// TIA Portal project "FactoryIO_Template_S7-1200_V15" (V15)
// Vorlageprojekt für das Buch mit Zielsystem S7-1200

(* hardware
DEVICE "S7-1200-Station_1"  S7-1200 Station
   slot 0: "Baugruppenträger_0"  Rack  V1.0
   slot 1: "PLC_1"  CPU 1211C DC/DC/DC  6ES7 211-1AE40-0XB0  V4.1
*)

// ===== PLC "PLC_1"  CPU 1211C DC/DC/DC =====

VAR_GLOBAL   // PLC tag table "Standard-Variablentabelle"
   "START" AT %I0.0 : Bool;
   "STOP" AT %I0.1 : Bool;
   "SENSOR 1" AT %I0.2 : Bool;
   "SENSOR 2" AT %I0.3 : Bool;
   "SENSOR 3" AT %I0.4 : Bool;
   "SENSOR 4" AT %I0.5 : Bool;
   "BELT 6m" AT %Q0.0 : Bool;
   "BELT 4m 1" AT %Q0.1 : Bool;
   "BELT 4m 2" AT %Q0.2 : Bool;
   "BELT 4m 3" AT %Q0.3 : Bool;
   "Wheel Right" AT %Q0.4 : Bool;
   "Wheel Left" AT %Q0.5 : Bool;
   "Wheel Forwerd" AT %Q0.6 : Bool;
   "Working" AT %Q0.7 : Bool;
   "Stoped" AT %Q1.0 : Bool;
   "X" AT %M0.0 : Bool;
   "Y" AT %M0.1 : Bool;
   "L" AT %M0.2 : Bool;
   "K" AT %M0.3 : Bool;
   "Tag_1" AT %M0.4 : Bool;
   "Tag_2" AT %M0.6 : Bool;
   "Tag_3" AT %M0.7 : Bool;
   "Tag_4" AT %M1.0 : Bool;
   "Tag_5" AT %M2.0 : Bool;
   "Tag_6" AT %M1.2 : Bool;
   "Tag_7" AT %M1.1 : Bool;
   "Tag_8" AT %M3.0 : Bool;
   "Tag_9" AT %M6.0 : Bool;
END_VAR

FUNCTION "MHJ-PLC-Lab-Function-S71200" : Void   // FC9000, SCL
{ S7_Optimized_Access := 'TRUE' }
VERSION : 0.1
   VAR_TEMP
      rdTimeReturn : Int;
      outputTime : DTL;
      SyncVal : Byte;
      forVal : Int;
      forVal_2 : Int;
      Value : Byte;
   END_VAR
   VAR CONSTANT
      CompVal : Byte := 16#34;
      Value_01 : Byte := 16#11;
      Value_01_DW : DWord := 16#A165_D992;
      Value_02_DW : DWord := 16#58BE_4401;
   END_VAR
BEGIN

   #Value:=PEEK(area := 16#82,
        dbNumber := 0,
        byteOffset := 511);
   #Value := #Value + 1;

   POKE(area := 16#82,
        dbNumber := 0,
        byteOffset := 511,
        value := #Value);

   POKE(area:=16#81,
        dbNumber:=0,
        byteOffset:=1016,
        value:=#Value_01_DW);
   POKE(area := 16#81,
        dbNumber := 0,
        byteOffset := 1020,
        value := #Value_02_DW);

   POKE(area := 16#81,
        dbNumber := 0,
        byteOffset := 511,
        value := B#16#00);

   FOR #forVal := 0 TO 120 DO
       FOR #forVal_2:=0 TO 10 DO
           #rdTimeReturn:=RD_SYS_T(#outputTime);
           #rdTimeReturn := WR_SYS_T(#outputTime);
           #rdTimeReturn := RD_SYS_T(#outputTime);
           #rdTimeReturn := WR_SYS_T(#outputTime);
       END_FOR;
       #SyncVal:= PEEK(area := 16#81,
                      dbNumber := 0,
                      byteOffset := 511);
       IF #SyncVal = #CompVal THEN
          GOTO M_1;
       END_IF;
   END_FOR;
   RETURN;

   M_1:
   POKE(area := 16#81,
        dbNumber := 0,
        byteOffset := 511,
        value := B#16#0);
END_FUNCTION

ORGANIZATION_BLOCK "Main"   // OB1, LAD, ProgramCycle
TITLE = "Main Program Sweep (Cycle)"
{ S7_Optimized_Access := 'TRUE' }
VERSION : 0.1
   VAR_INPUT
      Initial_Call : Bool;   // Initial call of this OB
      Remanence : Bool;   // =True, if remanent data are available
   END_VAR
   VAR_TEMP   // added for the SCL form of the ladder/FBD networks
      _w1 : Bool;
   END_VAR
BEGIN

REGION Network 1: Konnektierungsbaustein für PLC-Lab
   // Im Netzwerk 1 wird der Konnektierungsbaustein für PLC-Lab aufgerufen.
   // Dieser Aufruf darf nicht entfernt werden!
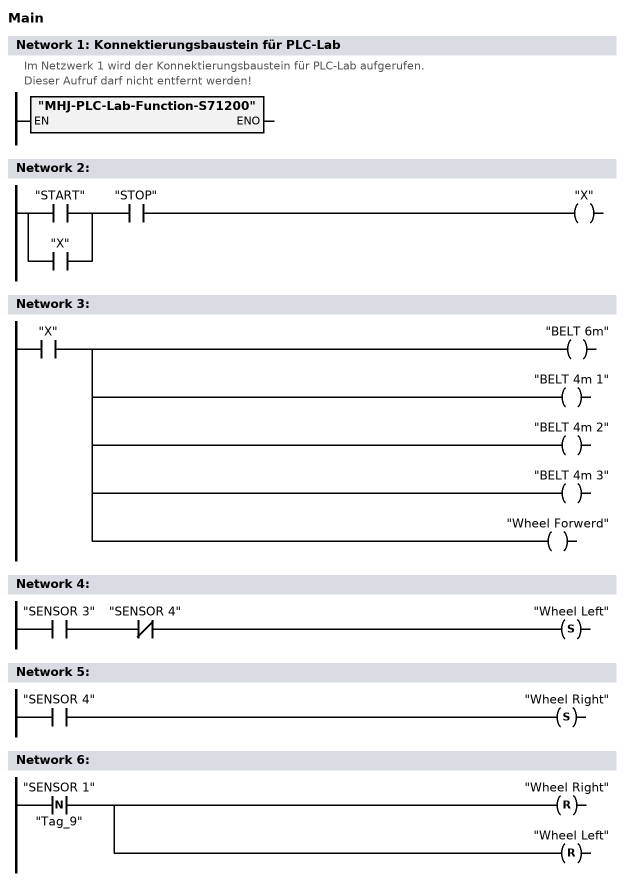
   RUNG wire#powerrail
      "MHJ-PLC-Lab-Function-S71200"()
   END_RUNG
   // the same network as SCL:
   "MHJ-PLC-Lab-Function-S71200"();
END_REGION

REGION Network 2
   RUNG wire#powerrail
      Contact( "START" )
      wire#w1
      Contact( "STOP" )
      Coil( "X" )
   END_RUNG
   RUNG wire#powerrail
      Contact( "X" )
   END_RUNG wire#w1
   // the same network as SCL:
   "X" := ("START" OR "X") AND "STOP";
END_REGION

REGION Network 3
   RUNG wire#powerrail
      Contact( "X" )
      wire#w1
      Coil( "BELT 6m" )
   END_RUNG
   RUNG wire#w1
      Coil( "BELT 4m 1" )
   END_RUNG
   RUNG wire#w1
      Coil( "BELT 4m 2" )
   END_RUNG
   RUNG wire#w1
      Coil( "BELT 4m 3" )
   END_RUNG
   RUNG wire#w1
      Coil( "Wheel Forwerd" )
   END_RUNG
   // the same network as SCL:
   "BELT 6m" := "X";
   "BELT 4m 1" := "X";
   "BELT 4m 2" := "X";
   "BELT 4m 3" := "X";
   "Wheel Forwerd" := "X";
END_REGION

REGION Network 4
   RUNG wire#powerrail
      Contact( "SENSOR 3" )
      I_Contact( "SENSOR 4" )
      S_Coil( "Wheel Left" )
   END_RUNG
   // the same network as SCL:
   IF "SENSOR 3" AND NOT "SENSOR 4" THEN "Wheel Left" := TRUE; END_IF;
END_REGION

REGION Network 5
   RUNG wire#powerrail
      Contact( "SENSOR 4" )
      S_Coil( "Wheel Right" )
   END_RUNG
   // the same network as SCL:
   IF "SENSOR 4" THEN "Wheel Right" := TRUE; END_IF;
END_REGION

REGION Network 6
   RUNG wire#powerrail
      N_Contact(operand := "SENSOR 1", bit := "Tag_9")
      wire#w1
      R_Coil( "Wheel Right" )
   END_RUNG
   RUNG wire#w1
      R_Coil( "Wheel Left" )
   END_RUNG
   // the same network as SCL:
   #_w1 := NOT "SENSOR 1" AND "Tag_9";   // falling edge of "SENSOR 1"
   "Tag_9" := "SENSOR 1";
   IF #_w1 THEN
       "Wheel Right" := FALSE;
       "Wheel Left" := FALSE;
   END_IF;
END_REGION
END_ORGANIZATION_BLOCK